PROGRAM P_Motion
VAR
	eAxis							:E_Axis;
	
	fbMcPowerTon					:ton;
	fbMcPowerREdge					:R_TRIG;
	fbMcPowerFEdge					:F_TRIG;
END_VAR

	//---各軸のステータスを読み込む---
	GVL.stAxis[E_Axis.X_Axis].ReadStatus();
	GVL.stAxis[E_Axis.Y_Axis].ReadStatus();
	GVL.stAxis[E_Axis.Z_Axis].ReadStatus();
	GVL.stAxis[E_Axis.Gripper].ReadStatus();
	
	//---各軸が動いているかをまとめる---
	GVL_Motion.bAxisMove:= GVL.stAxis[E_Axis.X_Axis].Status.Moving 
						OR GVL.stAxis[E_Axis.Y_Axis].Status.Moving
						OR GVL.stAxis[E_Axis.Z_Axis].Status.Moving 
						OR GVL.stAxis[E_Axis.Gripper].Status.Moving;
	
	//---マシンステートのファンクションブロックが停止出力していたら停止---
	GVL_Motion.bStop:=GVL_Alarm.fbMachineState.bStopMachine;

	//-----停止ボタン----
	GVL_Motion.bHalt:=GVL_MitsubishiCom.bFromMcHaltOn;
	
	//-----McPoerのOnとOff------
	fbMcPowerREdge(CLK:=GVL_MitsubishiCom.bFromMcPowerOn,Q=>);
	fbMcPowerFEdge(CLK:=GVL_MitsubishiCom.bToMcPowerOn,Q=>);
	fbMcPowerTon(IN:=GVL_MitsubishiCom.bFromMcPowerOn,PT:=T#3S,Q=>,ET=>);

	IF GVL_Motion.bPower=FALSE AND fbMcPowerREdge.Q=TRUE THEN;
		GVL_Motion.bPower:=TRUE;
	ELSIF GVL_Motion.bPower=TRUE AND fbMcPowerTon.Q=TRUE THEN ;
		GVL_Motion.bPower:=FALSE;
	ELSIF fbMcPowerFEdge.Q=TRUE THEN;
		GVL_Motion.bPower:=FALSE;
	END_IF;
	
	GVL_MitsubishiCom.bToMcPowerOn:= GVL_Motion.fbMcPower[E_Axis.X_Axis].Status
									AND GVL_Motion.fbMcPower[E_Axis.Y_Axis].Status 
									AND GVL_Motion.fbMcPower[E_Axis.Z_Axis].Status 
									AND GVL_Motion.fbMcPower[E_Axis.Gripper].Status;

	
	//-----ゼロポジション実行-----
	IF GVL_MitsubishiCom.bToMcPowerOn=TRUE THEN;
		GVL_Motion.bHome:=GVL_MitsubishiCom.bFromMcMoveHomeOn;
	END_IF
	
	GVL_MitsubishiCom.bToMcMoveHomeOn:=GVL_Motion.fbMcMoveHome[E_Axis.X_Axis].Busy
									OR GVL_Motion.fbMcMoveHome[E_Axis.Y_Axis].Busy
									OR GVL_Motion.fbMcMoveHome[E_Axis.Z_Axis].Busy
									OR GVL_Motion.fbMcMoveHome[E_Axis.Gripper].Busy;

	//-----Jog実行-----
	IF GVL_MitsubishiCom.bToMcPowerOn=TRUE THEN;
		//X軸
		GVL_Motion.bJog[E_Axis.X_Axis]:=GVL_MitsubishiCom.bFromXAxisJogStart;
		GVL_Motion.lrJogPosition[E_Axis.X_Axis]:=GVL_MitsubishiCom.wFromXAxisJogTarget;
		
		//Y軸
		GVL_Motion.bJog[E_Axis.Y_Axis]:=GVL_MitsubishiCom.bFromYAxisJogStart;
		GVL_Motion.lrJogPosition[E_Axis.Y_Axis]:=GVL_MitsubishiCom.wFromYAxisJogTarget;
		
		//Z軸 ステージにグリッパーがあたるのでZ軸は300無しで
		GVL_Motion.bJog[E_Axis.Z_Axis]:=GVL_MitsubishiCom.bFromZAxisJogStart;
		GVL_Motion.lrJogPosition[E_Axis.Z_Axis]:=GVL_MitsubishiCom.wFromZAxisJogTarget;
		IF GVL_Motion.lrJogPosition[E_Axis.Z_Axis]>230 THEN;
			GVL_Motion.lrJogPosition[E_Axis.Z_Axis]:=225;
		END_IF

		//グリッパー
		GVL_Motion.bJog[E_Axis.Gripper]:=GVL_MitsubishiCom.bFromGripperJogStart;
		GVL_Motion.lrJogPosition[E_Axis.Gripper]:=WORD_TO_INT(GVL_MitsubishiCom.wFromGripperJogTarget);
	END_IF
	
	//---アクションをコールして軸を起動---
	FOR eAxis:= E_Axis.X_Axis TO E_Axis.Gripper DO
		aMotion();
	END_FOR;

ACTION aMotion:
//パワーON
	GVL_Motion.fbMcPower[eAxis](
		Axis			:=GVL.stAxis[eAxis],
		Enable			:=GVL_Motion.bPower,
		Enable_Positive	:=GVL_Motion.bPower,
		Enable_Negative	:=GVL_Motion.bPower,
		Override		:=100,
		Status			=>,
		Busy			=>,
		Active			=>,
		Error			=>,
		ErrorID			=>
	);
	
//ホーミング
	GVL_Motion.fbMcMoveHome[eAxis](
		Axis			:=GVL.stAxis[eAxis],
		Execute			:=GVL_Motion.bHome,
		Position		:=0,
		Velocity		:=50,
		Done			=>,
		Busy			=>,
		Active			=>,
		CommandAborted	=>,
		Error			=>,
		ErrorID			=>
	);	

//ジョグ
	GVL_Motion.fbMcMoveJog[eAxis](
		Axis			:=GVL.stAxis[eAxis],
		Execute			:=GVL_Motion.bJog[eAxis],
		Position		:=GVL_Motion.lrJogPosition[eAxis],
		Velocity		:=50,
		Done			=>,
		Busy			=>,
		Active			=>,
		CommandAborted	=>,
		Error			=>,
		ErrorID			=>
	);	
	
//全軸一時停止
	GVL_Motion.fbMCHalt[eAxis](
		Axis			:=GVL.stAxis[eAxis],
		Execute			:=GVL_Motion.bHalt,
		Done			=>,
		Busy			=>,
		Active			=>,
		CommandAborted	=>,
		Error			=>,
		ErrorID			=>
	);

//全軸ストップ
	GVL_Motion.fbMCStop[eAxis](
		Axis			:=GVL.stAxis[eAxis],
		Execute			:=GVL_Motion.bStop,
		Done			=>,
		Busy			=>,
		Active			=>,
		CommandAborted	=>,
		Error			=>,
		ErrorID			=>
	);
	
//全軸リセット
	GVL_Motion.fbMcReset[eAxis](
		Axis			:=GVL.stAxis[eAxis],
		Execute			:=GVL_Motion.bReset,
		Done			=>,
		Busy			=>,
		Error			=>,
		ErrorID			=>
	);
END_ACTION

END_PROGRAM

(* stored: Version 1.1.0.1, ProductVersion 3.1.4024.12
   POU P_Motion: Id {f27a55a5-997f-454a-b871-3cb76ed937db}, SpecialFunc None
   Action aMotion: Id {7128f73f-11b3-4c17-add6-4b6df319662d} *)
